TYPE ST_GantryXYZ_Command :
    STRUCT
	
    END_STRUCT
END_TYPE

(* stored: Version 1.1.0.1, ProductVersion 3.1.4024.15
   DUT ST_GantryXYZ_Command: Id {006df9d5-63c6-42f0-b149-eff97f907bc4} *)
